Staubli VAL3: getFunctionEdit.pgx

public program getFunctionEdit(string& x_sName[])
begin
  //
  // define your message for the
  // function KEY
  //
  // NOTE is an ARRAY[0..7]
  //
  // example:
  // x_sName[1]="DEMO"
  // active the F2 button
  //
end
